PROGRAM TanksSimulation
VAR_INPUT
	bStart AT %I* : BOOL;
	bEmerNC AT %I*: BOOL;
	bHI AT %I*: BOOL;
	bLO AT %I*: BOOL;
END_VAR	
VAR_OUTPUT
	bMotor1 AT %Q*: BOOL;
	bMotor2 AT %Q*: BOOL;
	bRun AT %Q*: BOOL;
	bErr AT %Q*: BOOL;
END_VAR
VAR
	bStateOn: BOOL := FALSE;
	bStateErr: BOOL := FALSE;
	trigStateOn: R_TRIG;
	bFirstScan: BOOL;
END_VAR

trigStateOn(CLK:= bStart);
IF trigStateOn.Q THEN
	IF bStateOn THEN
		bStateOn := FALSE;
	ELSE
		bStateOn := TRUE;
		bStateErr := FALSE;
		bMotor2 := TRUE;
	END_IF
END_IF

IF NOT bEmerNC THEN
	bStateErr := TRUE;
	bStateOn := FALSE;
END_IF

IF bStateOn THEN 
	IF NOT bHI THEN
		bMotor1:= FALSE;
		bMotor2:= TRUE;
	END_IF
	
	IF bLO THEN
		bMotor1:= TRUE;
		bMotor2:= FALSE;
	END_IF
ELSE
	bMotor1:= FALSE;
	bMotor2:= FALSE;
END_IF

bRun := bStateOn;
bErr := bStateErr;

END_PROGRAM

(* stored: Version 1.1.0.1, ProductVersion 3.1.4024.4
   POU TanksSimulation: Id {c46e3ad6-3c2c-4e43-9ba2-dcd67fb724f8}, SpecialFunc None *)
